FUNCTION F_Concat4 : T_MaxString
VAR_INPUT
	sOne 	: STRING;
	sTwo	: STRING;
	sThree	: STRING;
	sFour	: STRING;
END_VAR

F_Concat4 := CONCAT(
					sOne,
					F_Concat3( sTwo, sThree, sFour )
				);

END_FUNCTION

(* stored: Version 1.1.0.1, ProductVersion 3.1.4022.9
   POU F_Concat4: Id {89dab43a-8967-46e8-aa27-51cc7be08d74}, SpecialFunc None *)
